PROGRAM Fast_Faults_Evaluate
VAR

END_VAR

g_FastFaultOutput2.EvaluateOutput(bAutoReset:=TRUE);

END_PROGRAM

(* stored: Version 1.1.0.1, ProductVersion 3.1.4022.18
   POU Fast_Faults_Evaluate: Id {667ad34f-81ff-0404-3362-bb63097d9547}, SpecialFunc None *)
